Staubli VAL3: ExtraAxis.pgx

public program ExtraAxis()
begin

  //如果七轴当前位置与所需位置不一致
  //if
  //bExtraAxis
  waitEndMove()


  //让七轴运动起来

  //wait 七轴位置到位

  //end






end
